Universal Robots PolyScope program: attention_to_human.urp

Program attention_to_human (installation=default directory=/home/ur/ursim-current/programs createdIn=3.14.1.1031110 lastSavedIn=3.14.1.1031110 robotSerialNumber=2018309999)
Calibrated DH parameters: a=[0, -0.612, -0.5723, 0, 0, 0]; d=[0.1273, 0, 0, 0.163941, 0.1157, 0.0922]; alpha=[1.570796, 0, 0, 1.570796, -1.570796, 0]; deltaTheta=[0, 0, 0, 0, 0, 0]
Robot Program (runOnlyOnce=false)
  MoveJ speed 60 deg/s, acceleration 80 deg/s^2 (useActiveTCP=true)
    Waypoint Waypoint_1: TCP in base x=281.272 y=-152.342 z=230.789 mm, rx=-0.0012 ry=3.1163 rz=0.0389 rad; joints [1.928, -60.308, -156.017, -52.191, 91.381, 91.901] deg
    Waypoint Waypoint_2: TCP in base x=284.266 y=-152.242 z=938.568 mm, rx=-0.0172 ry=1.8569 rz=0.0688 rad; joints [1.928, -53.484, -102.341, -40.543, 91.381, 91.901] deg
    Wait Sleep waitTime=3
